PROGRAM MAIN
VAR
	lrIn AT%I* : LREAL := 0;
	nCheckCount : INT := 0;
	
	fbPlantNo1: PlantNo1;
	fbPlantNo2: PlantNo2;
	lrOutput AT%Q* : LREAL := 0.0;
	
	nPlant :INT := 0;
	
	lrTempOutput : LREAL := 0.0;
	
	
END_VAR

CASE nPlant OF
	10:
		fbPlantNo1(lrInput := lrIn,
		lrOutput => lrOutput);
		
	20:
		fbPlantNo2(lrInput := lrIn,
			lrM := 3.5,
			lrC := 10,
		lrOutput => lrOutput);
		
	30:
		fbPlantNo1(lrInput := lrIn,
			lrOutput => lrTempOutput);
		fbPlantNo2(lrInput := lrTempOutput,
			lrM := 3.5,
			lrC := 10,
			lrOutput => lrOutput);
			
END_CASE

END_PROGRAM

(* stored: Version 1.1.0.1, ProductVersion 3.1.4026.8
   POU MAIN: Id {65c70385-e05c-4e29-a597-92e55abc482c}, SpecialFunc None *)
